Yaskawa INFORM job: R1_W08,11(-70,-90)_KM-OK.JBI

/JOB
//NAME R1_W08,11(-70,-90)_KM-OK
///FOLDERNAME KRIS-SCIANA
//POS
///NPOS 79,79,0,3,0,0
///TOOL 0
///POSTYPE PULSE
///PULSE
C00000=-80634,56423,27720,33300,115319,-48613
C00001=-80634,56524,26439,33552,116027,-48375
C00002=-80628,58269,45036,31008,107028,-51169
C00003=-78911,55316,44053,31183,105606,-50866
C00004=-78212,54208,43755,31252,105015,-50747
C00005=-78077,53876,44572,31170,104384,-50872
C00006=-78212,54208,43755,31252,105015,-50747
C00007=-75675,58994,46299,31860,104831,-49753
C00008=-75090,60550,48062,31915,104366,-49647
C00009=-75675,58994,46299,31860,104831,-49753
C00010=-73415,47128,27098,33303,108822,-47587
C00011=-73012,45246,24655,33476,109116,-47321
C00012=-73415,47128,27098,33303,108822,-47587
C00013=-74150,48191,27319,33287,109454,-47700
C00014=-75960,51015,28077,33247,110987,-47988
C00015=-75965,52987,13601,36257,119226,-45094
C00016=-136517,51935,5119,1923,104393,-8731
C00017=-87157,-5483,-28306,-57450,115604,-41571
C00018=-87147,-5039,-11335,-53427,109619,-37333
C00019=-88649,-5898,-8462,-52940,107396,-36805
C00020=-89258,-6153,-7236,-52774,106498,-36599
C00021=-87889,14537,19903,-58993,114209,-37793
C00022=-88767,13530,18983,-59246,113694,-37990
C00023=-87889,14537,19903,-58993,114209,-37793
C00024=-87649,13613,19920,-58714,114095,-37532
C00025=-87889,14537,19903,-58993,114209,-37793
C00026=-105942,-62521,-63510,-26568,80862,-38232
C00027=-105031,-65851,-62417,-26893,79012,-37461
C00028=-105195,-64382,-61180,-26864,78954,-37510
C00029=-105031,-65851,-62417,-26893,79012,-37461
C00030=-105431,-67258,-67024,-26678,80780,-38021
C00031=-107641,-43424,-69167,-26047,92329,-41409
C00032=-143143,24328,-21242,15658,96224,11878
C00033=-72204,74256,59569,26405,111997,-60927
C00034=-70917,68999,55676,26710,111311,-60566
C00035=-85864,57700,53549,32032,120643,-64746
C00036=-70563,68474,57156,26581,110137,-60710
C00037=-70776,68944,56037,26701,111041,-60575
C00038=-82327,65803,62898,33102,117932,-64007
C00039=-66932,87982,79688,30579,103155,-62915
C00040=-68273,94194,85253,30231,103438,-63379
C00041=-67652,72456,53103,19372,121960,-51858
C00042=-68730,81297,71878,24437,120905,-53913
C00043=-70977,68393,57703,23430,124019,-52775
C00044=-66315,67012,49556,19800,121060,-51456
C00045=-65775,67263,51320,19811,120027,-51426
C00046=-73586,65272,57175,21672,123548,-54069
C00047=-68991,63069,47524,18483,120952,-52622
C00048=-70206,68275,51151,18045,121645,-53017
C00049=-67306,51124,50401,20344,101560,-40970
C00050=-87477,30209,35148,22218,113002,-46164
C00051=-84814,33924,44185,23054,109360,-46670
C00052=-65224,53044,56715,20613,98319,-40767
C00053=-65298,47795,50229,20686,99552,-40580
C00054=-87988,42110,60194,20988,104936,-48724
C00055=-71908,43018,52479,24041,92531,-45521
C00056=-73734,43279,49847,23760,94663,-45760
C00057=-75710,44802,35372,24197,104128,-44564
C00058=-131785,47166,14001,6017,108119,-46057
C00059=-158927,32103,13676,-68669,79329,-67442
C00060=-158908,36411,34815,-70732,75312,-62704
C00061=-161041,36978,37858,-71079,73298,-62259
C00062=-161585,38964,41701,-71458,72462,-61721
C00063=-161197,36103,37872,-71200,73031,-62071
C00064=-161616,38399,39420,-71134,72825,-62225
C00065=-159919,52811,61984,-72937,71813,-59077
C00066=-159331,51665,59666,-72650,72481,-59393
C00067=-153527,56458,59991,-71753,77181,-59746
C00068=-155097,66673,45520,-46808,107874,38774
C00069=-160646,74114,58732,-46422,101973,38891
C00070=-161246,72438,57080,-46511,101769,38689
C00071=-160874,72062,56896,-46460,101906,38810
C00072=-161157,75917,61015,-46390,101370,38929
C00073=-162992,77000,64707,-38887,97568,39674
C00074=-159778,86810,81631,-45169,97042,41627
C00075=-157799,88241,81814,-44919,98490,41911
C00076=-156482,94558,73923,-46181,104945,39526
C00077=-167679,39598,-22082,-19335,97230,42029
C00078=-169349,-60111,-118624,-3020,75160,29230
BC00000=67240,746139,887723
BC00001=876,746139,637498
BC00002=876,746139,637498
BC00003=876,746139,637498
BC00004=876,746139,637498
BC00005=876,746139,637498
BC00006=876,746139,637498
BC00007=876,746139,637498
BC00008=876,746139,637498
BC00009=876,746139,637498
BC00010=876,746139,637498
BC00011=876,746139,637498
BC00012=876,746139,637498
BC00013=876,746139,637498
BC00014=876,746139,637498
BC00015=876,746139,637498
BC00016=162851,665976,600131
BC00017=75688,710588,698134
BC00018=75688,710588,698134
BC00019=75688,710588,698134
BC00020=75688,710588,698134
BC00021=75688,710588,698134
BC00022=75688,710588,698134
BC00023=75688,710588,698134
BC00024=75688,710588,698134
BC00025=75688,710588,698134
BC00026=75688,710588,698134
BC00027=75688,710588,698134
BC00028=75688,710588,698134
BC00029=75688,710588,698134
BC00030=75688,710588,698134
BC00031=75688,710588,698134
BC00032=162851,669294,600131
BC00033=19061,743600,675276
BC00034=19061,743600,675276
BC00035=65065,743601,675267
BC00036=19061,743600,675276
BC00037=19061,743600,675276
BC00038=77929,743601,675267
BC00039=19061,743600,675276
BC00040=19061,743600,675276
BC00041=27646,753773,647623
BC00042=27646,753773,647623
BC00043=40792,753773,647623
BC00044=27646,753773,647623
BC00045=27646,753773,647623
BC00046=40792,753773,647623
BC00047=27646,753773,647623
BC00048=27646,753773,647623
BC00049=8546,760690,801679
BC00050=69038,760690,801679
BC00051=65023,760690,801679
BC00052=8546,760690,801679
BC00053=8546,760690,801679
BC00054=65023,760690,801679
BC00055=8546,760690,801679
BC00056=8546,760690,801679
BC00057=8546,760690,801679
BC00058=126110,665470,679172
BC00059=279808,708395,661827
BC00060=279808,708395,661827
BC00061=279808,708395,661827
BC00062=279807,708393,661826
BC00063=279808,708395,661827
BC00064=279808,708395,661827
BC00065=279808,708395,661827
BC00066=279808,708395,661827
BC00067=279808,708395,661827
BC00068=260779,714461,579821
BC00069=260779,714461,579821
BC00070=260779,714461,579821
BC00071=260779,714461,579821
BC00072=260779,714461,579821
BC00073=260779,714461,579821
BC00074=260779,714461,579821
BC00075=260779,714461,579821
BC00076=260779,714461,579821
BC00077=260780,714460,579818
BC00078=240210,673556,584383
///POSTYPE BASE
///RECTAN
///RCONF 0,0,0,0,0,0,0,0,0,0,0,0,0,0,0,0,0,0,0,0,0,0,0,0
P00006=0.222,-3.123,-1.508,0.0000,0.0000,0.0000
P00021=-0.225,-6.128,-0.405,0.0000,0.0000,0.0000
P00026=0.562,-0.002,-0.337,0.0000,0.0000,0.0000
//INST
///DATE 2024/07/23 15:33
///ATTR SC,RW
///GROUP1 RB1,BS1
NOP
'r2_W08,11(-70,-90)
'Path S787 (for W8)
SFTOF
MOVJ C00000 BC00000 VJ=100.00
MOVJ C00001 BC00001 VJ=50.00
MOVJ C00002 BC00002 VJ=100.00
MOVL C00003 BC00003 V=100.0
MOVL C00004 BC00004 V=60.0
REFP 3 C00005 BC00005
CALL JOB:SEARCH-R1
SET P021 P006
SFTON P021
MOVL C00006 BC00006 V=60.0
MOVL C00007 BC00007 V=60.0
REFP 3 C00008 BC00008
CALL JOB:SEARCH-R1
SET P021 P006
SFTON P021
MOVL C00009 BC00009 V=60.0
MOVL C00010 BC00010 V=60.0
REFP 3 C00011 BC00011
CALL JOB:SEARCH-R1
SET P021 P006
SFTON P021
MOVL C00012 BC00012 V=133.3
MOVL C00013 BC00013 V=250.0
MOVL C00014 BC00014 V=250.0
MOVL C00015 BC00015 V=250.0
MOVJ C00016 BC00016 VJ=100.00
'Path S867
SFTOF
MOVJ C00017 BC00017 VJ=100.00
MOVJ C00018 BC00018 VJ=100.00
MOVL C00019 BC00019 V=250.0
MOVL C00020 BC00020 V=250.0
MOVL C00021 BC00021 V=133.3
REFP 3 C00022 BC00022
CALL JOB:SEARCH-R1
SET P026 P006
SFTON P026
MOVL C00023 BC00023 V=133.3
REFP 3 C00024 BC00024
CALL JOB:SEARCH-R1
SET P026 P006
SFTON P026
MOVL C00025 BC00025 V=166.7
MOVL C00026 BC00026 V=166.7
MOVL C00027 BC00027 V=166.7
REFP 3 C00028 BC00028
CALL JOB:SEARCH-R1
SET P026 P006
SFTON P026
MOVL C00029 BC00029 V=166.7
MOVL C00030 BC00030 V=500.0
MOVL C00031 BC00031 V=1000.0
MOVJ C00032 BC00032 VJ=100.00
'Path W5
SFTOF
SFTON P021
MOVJ C00033 BC00033 VJ=100.00
MOVL C00034 BC00034 V=100.0
MOVL C00035 BC00035 V=166.7 PL=0
REFP 1 C00036 BC00036
REFP 2 C00037 BC00037
MACRO1 MJ#(0) ARGF6
ARCON
MOVL C00038 BC00038 V=8.3
ARCOF
MOVL C00039 BC00039 V=100.0
MOVL C00040 BC00040 V=100.0
SFTOF
'Path W6
SFTOF
SFTON P021
MOVJ C00041 BC00041 VJ=100.00
MOVL C00042 BC00042 V=100.0
MOVL C00043 BC00043 V=100.0 PL=0
REFP 1 C00044 BC00044
REFP 2 C00045 BC00045
MACRO1 MJ#(0) ARGF6
ARCON
MOVL C00046 BC00046 V=8.3
ARCOF
MOVL C00047 BC00047 V=100.0
MOVL C00048 BC00048 V=100.0
SFTOF
'Path W7
SFTOF
SFTON P021
MOVJ C00049 BC00049 VJ=100.00
MOVL C00050 BC00050 V=333.3
MOVL C00051 BC00051 V=166.7 PL=0
REFP 1 C00052 BC00052
REFP 2 C00053 BC00053
MACRO1 MJ#(0) ARGF6
ARCON
MOVL C00054 BC00054 V=8.3
ARCOF
MOVL C00055 BC00055 V=100.0
MOVL C00056 BC00056 V=100.0
MOVL C00057 BC00057 V=100.0
SFTOF
MOVJ C00058 BC00058 VJ=100.00
'
'Path W8
SFTOF
SFTON P026
MOVJ C00059 BC00059 VJ=100.00
MOVJ C00060 BC00060 VJ=100.00
MOVL C00061 BC00061 V=250.0
MOVL C00062 BC00062 V=166.7 PL=0
REFP 1 C00063 BC00063
REFP 2 C00064 BC00064
MACRO1 MJ#(0) ARGF6
ARCON
MOVL C00065 BC00065 V=8.3
ARCOF
MOVL C00066 BC00066 V=250.0
MOVJ C00067 BC00067 VJ=100.00
SFTOF
'Path W868
SFTOF
SFTON P026
MOVJ C00068 BC00068 VJ=100.00
MOVL C00069 BC00069 V=250.0
MOVL C00070 BC00070 V=166.7 PL=0
REFP 1 C00071 BC00071
REFP 2 C00072 BC00072
MACRO1 MJ#(0) ARGF6
ARCON
MOVL C00073 BC00073 V=8.3
ARCOF
MOVL C00074 BC00074 V=166.7
MOVL C00075 BC00075 V=250.0
MOVL C00076 BC00076 V=333.3
SFTOF
MOVJ C00077 BC00077 VJ=100.00
MOVJ C00078 BC00078 VJ=100.00
END
